SUBAPPLICATION RegsiterEmergencyLight (* Subapplication Type *)
  (* Standard: 61499-2 *)
  (* Version 1.0, 2018-11-28, cabral *)
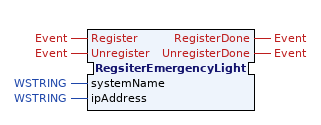
  EVENT_INPUT
    Register;
    Unregister;
  END_EVENT
  EVENT_OUTPUT
    RegisterDone;
    UnregisterDone;
  END_EVENT
  VAR_INPUT
    systemName : WSTRING := WSTRING#wsnGateway144-mediator-0;
    ipAddress : WSTRING := WSTRING#%localIP%;
  END_VAR
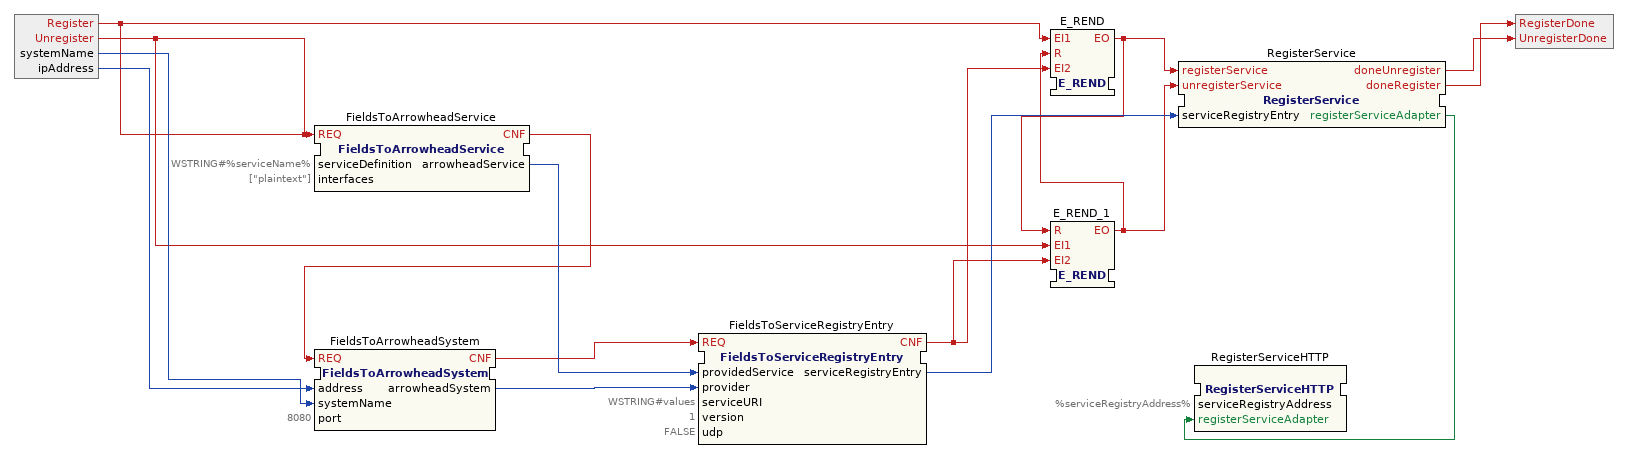
  FBS
    FieldsToArrowheadService : FieldsToArrowheadService(serviceDefinition := WSTRING#%serviceName%, interfaces := ["plaintext"]);
    FieldsToArrowheadSystem : FieldsToArrowheadSystem(port := 8080);
    RegisterServiceHTTP : RegisterServiceHTTP(serviceRegistryAddress := %serviceRegistryAddress%);
    E_REND : E_REND;
    E_REND_1 : E_REND;
    RegisterService : RegisterService;
    FieldsToServiceRegistryEntry : FieldsToServiceRegistryEntry(serviceURI := WSTRING#values, version := 1, udp := FALSE);
  END_FBS
  EVENT_CONNECTIONS
    FieldsToArrowheadService.CNF TO FieldsToArrowheadSystem.REQ;
    Register TO FieldsToArrowheadService.REQ;
    Unregister TO FieldsToArrowheadService.REQ;
    Register TO E_REND.EI1;
    E_REND_1.EO TO E_REND.R;
    E_REND.EO TO E_REND_1.R;
    Unregister TO E_REND_1.EI1;
    E_REND.EO TO RegisterService.registerService;
    E_REND_1.EO TO RegisterService.unregisterService;
    RegisterService.doneUnregister TO UnregisterDone;
    RegisterService.doneRegister TO RegisterDone;
    FieldsToServiceRegistryEntry.CNF TO E_REND_1.EI2;
    FieldsToServiceRegistryEntry.CNF TO E_REND.EI2;
    FieldsToArrowheadSystem.CNF TO FieldsToServiceRegistryEntry.REQ;
  END_CONNECTIONS
  DATA_CONNECTIONS
    ipAddress TO FieldsToArrowheadSystem.address;
    systemName TO FieldsToArrowheadSystem.systemName;
    FieldsToArrowheadService.arrowheadService TO FieldsToServiceRegistryEntry.providedService;
    FieldsToArrowheadSystem.arrowheadSystem TO FieldsToServiceRegistryEntry.provider;
    FieldsToServiceRegistryEntry.serviceRegistryEntry TO RegisterService.serviceRegistryEntry;
  END_CONNECTIONS
  ADAPTER_CONNECTIONS
    RegisterService.registerServiceAdapter TO RegisterServiceHTTP.registerServiceAdapter;
  END_CONNECTIONS
END_SUBAPPLICATION
